INTERFACE I_Notification

METHOD AddNotificationHandler : I_Notification
VAR_INPUT
    Handler : I_NotificationHandler;
END_VAR
END_METHOD

PROPERTY Args : I_StreamWriter
GET
END_GET
END_PROPERTY

METHOD ClearNotificationHandlers : I_Notification
VAR_INPUT
END_VAR
END_METHOD

METHOD Raise
END_METHOD

END_INTERFACE

(* stored: Version 1.1.0.1, ProductVersion 3.1.4024.9
   Itf I_Notification: Id {7718dd74-9654-4af8-a63b-c5e9a3756592}
   Folder Methods: Id {934cf189-59cc-432d-80de-bb374f150b04}
   Folder Properties: Id {f693607d-d6ad-4277-ac98-609e275d0af6}
   Method AddNotificationHandler: Id {a599c9f3-32fa-4f0e-9ef6-b5a88dd029bc}
   Property Args: Id {404a8398-597e-4d06-b5b1-3cad519ea9d9}
   Get Get: Id {191e915c-188e-4375-a4cb-7d82d278b82a}
   Method ClearNotificationHandlers: Id {aae0fbce-130c-410d-913a-232b8d930f74}
   Method Raise: Id {39bb1e56-1c4d-4d8d-9ff2-78ad891a1fca} *)
